SUBAPPLICATION Uebung_011 (* Numeric Value Input *)
  (* Standard: 61499-2; Description: Copyright (c) 2023 Meisterschulen am Ostbahnhof This program and the accompanying materials are made available under the terms of the Eclipse Public License 2.0 which is available at https://www.eclipse.org/legal/epl-2.0/ SPDX-License-Identifier: EPL-2.0 *)
  (* Version 1.0, 2023-10-23, Franz Höpfinger, Meisterschulen am Ostbahnhof *)
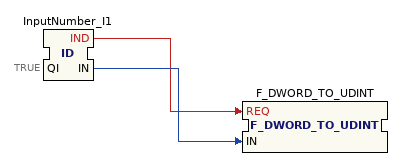
  FBS
    F_DWORD_TO_UDINT : F_DWORD_TO_UDINT;
    InputNumber_I1 : ID(QI := TRUE);
  END_FBS
  EVENT_CONNECTIONS
    InputNumber_I1.IND TO F_DWORD_TO_UDINT.REQ;
  END_CONNECTIONS
  DATA_CONNECTIONS
    InputNumber_I1.IN TO F_DWORD_TO_UDINT.IN;
  END_CONNECTIONS
END_SUBAPPLICATION
